{attribute 'qualified_only'}
{attribute 'strict'}
TYPE E_ViseSocketState :
(
	ViseInSocket := 0,
	SocketEmpty	:= 1
);
END_TYPE

(* stored: Version 1.1.0.1, ProductVersion 3.1.4024.12
   DUT E_ViseSocketState: Id {6f7f6291-4493-49de-b400-0fde49631d3c} *)
